// TIA Portal V16 export
// export: Created 2025-08-01T13:38:14.4676832Z, ExportSetting WithDefaults, DisplayName Totally Integrated Automation Portal, DisplayVersion V16, DisplayName TIA Portal Version Control Interface, DisplayVersion V16, DisplayName TIA Portal Openness, DisplayVersion V16, DisplayName STEP 7 Professional, DisplayVersion V16, DisplayName STEP 7 Safety, DisplayVersion V16, DisplayName WinCC Advanced, DisplayVersion V16
VAR_GLOBAL   // PLC tag table "Default tag table"
   "Drive 1 Ready" AT %I0.0 : Bool;   // +MC-21K2:1 - Drive 1 Ready
   "Drive 2 Ready" AT %I0.1 : Bool;   // +MC-21K2:5 - Drive 2 Ready
   "Drive 3 Ready" AT %I0.2 : Bool;   // +MC-21K2:2 - Drive 3 Ready
   "Drive 4 Ready" AT %I0.3 : Bool;   // +MC-21K2:6 - Drive 4 Ready
   "Drive 5 Ready" AT %I0.4 : Bool;   // +MC-21K2:3 - Drive 5 Ready
   "Sensor Trechter" AT %I0.5 : Bool;   // +MC-21K2:7 - Sensor Trechter
   "Sensor Op Band" AT %I0.6 : Bool;   // +MC-21K2:4 Sensor Op Band
   "Sensor Wals (Option)" AT %I0.7 : Bool;   // +MC-21K2:8 - Sensor Wals (Option)
   "ESB Oke" AT %I1.0 : Bool;   // +MC-21K3:1 - ESB Oke
   "ESB Pressend" AT %I1.1 : Bool;   // +MC-21K3:5 - ESB Pressend
   "Reset Active" AT %I1.2 : Bool;   // +MC-21K3:2 - Reset Active
   "Noodsleutel(1)" AT %I1.3 : Bool;   // +MC-21K3:6 - NOODSLEUTEL
   "Alle uitgangen(1)" AT %I1.4 : Bool;   // +MC-21K3:3 - Alle uitgangen
   "Door 1 NC contact" AT %I1.5 : Bool;   // +MC-21K3:7 - Safety Doorswitch 1
   "Door 1 NO contact" AT %I1.6 : Bool;   // +MC-21K3:4 - Safety Doorswitch 1 Normaly open
   "Door 2 NC contact" AT %I1.7 : Bool;   // +MC-21K3:8 - Safety Doorswitch 2
   "Spare(5)" AT %I3.0 : Bool;
   "Spare(6)" AT %I3.1 : Bool;
   "Spare(10)" AT %I180.0 : Bool;   // Spare
   "Spare(11)" AT %I180.1 : Bool;   // Spare
   "Spare(12)" AT %I3.4 : Bool;   // Spare
   "Spare(13)" AT %I3.5 : Bool;   // Spare
   "Spare(14)" AT %I3.6 : Bool;   // Spare
   "Spare(15)" AT %I3.7 : Bool;   // Spare
   "Programma 1" AT %I2.0 : Bool;   // +MC-21K4:1 - Programma 1
   "Programma 2" AT %I2.1 : Bool;   // +MC-21K4:5 - Programma 2 (Option)
   "Programma 3" AT %I2.2 : Bool;   // +MC-21K4:2 - Programma 3
   Cleaning AT %I2.3 : Bool;   // +MC-21K4:6 - Cleaning
   "Start Machine" AT %I2.4 : Bool;   // +MC-21K4:3 - Start Machine
   "Stop Machine" AT %I2.5 : Bool;   // +MC-21K4:7 - Stop Machine
   "Spare(16)" AT %I2.6 : Bool;   // Spare
   Encoder_Z_Puls AT %I2.7 : Bool;   // Spare
   "Safety Relais" AT %Q0.0 : Bool;   // +MC-21K6:1 - Safety Relais
   "Bel Storing" AT %Q0.1 : Bool;   // +MC-21K6:5 - Bel Storing
   Spare AT %Q5.3 : Bool;   // Spare
   "Drive 1 RUN FWD" AT %Q1.0 : Bool;   // +MC-21K8:1 - Drive 1 RUN FWD
   "Drive 1 REV]" AT %Q1.1 : Bool;   // +MC-21K8:5 - Drive 1 REV
   "Drive 1 Speed 1" AT %Q1.2 : Bool;   // +MC-21K8:2 - Drive 1 Speed 1
   "Drive 1 Speed 2" AT %Q1.3 : Bool;   // +MC-21K8:6 - Drive 1 Speed 2
   "Spare(3)" AT %Q1.4 : Bool;   // Spare
   "Drive 2 RUN FWD" AT %Q1.5 : Bool;   // +MC-21K8:7 - Drive 2 RUN FWD
   "Drive 2 REV" AT %Q1.6 : Bool;   // +MC-21K8:4 - Drive 2 REV
   "Drive 2 Speed 1" AT %Q1.7 : Bool;   // +MC-21K8:8 - Drive 2 Speed 1
   "Drive 2 Speed 2" AT %Q2.0 : Bool;   // +MC-21K9:1 - Drive 2 Speed 2
   "Spare(4)" AT %Q2.1 : Bool;   // Spare
   "Drive 3 RUN FWD" AT %Q2.2 : Bool;   // +MC-21K9:2 - Drive 3 RUN FWD
   "Drive 3 REV" AT %Q2.3 : Bool;   // +MC-21K9:6 - Drive 3 REV
   "Drive 3 Speed 1" AT %Q2.4 : Bool;   // +MC-21K9:3 - Drive 3 Speed 1
   "Drive 3 Speed 2" AT %Q2.5 : Bool;   // +MC-21K9:7 - Drive 3 Speed 2
   "Spare(21)" AT %Q2.6 : Bool;   // Spare
   "Drive 4 RUN FWD" AT %Q2.7 : Bool;   // +MC-21K9:8 - Drive 4 RUN FWD
   "Drive 4 REV" AT %Q3.0 : Bool;   // +MC-21K10:1 - Drive 4 REV
   "Drive 4 Speed 1" AT %Q3.1 : Bool;   // +MC-21K10:5 - Drive 4 Speed 1
   "Drive 4 Speed 2" AT %Q3.2 : Bool;   // +MC-21K10:2 - Drive 4 Speed 2
   "Spare(22)" AT %Q3.3 : Bool;   // Spare
   "Drive 5 RUN FWD" AT %Q3.4 : Bool;   // +MC-21K10:3 - Drive 5 RUN FWD
   "Drive 5 REV" AT %Q3.5 : Bool;   // +MC-21K10:7 - Drive 5 REV
   "Drive 5 Speed 1" AT %Q3.6 : Bool;   // +MC-21K10:4 - Drive 5 Speed 1
   "Drive 5 Speed 2" AT %Q3.7 : Bool;   // +MC-21K10:8 - Drive 5 Speed 2
   "Spare(23)" AT %Q4.0 : Bool;   // Spare
   "LED Programma 1" AT %Q4.1 : Bool;   // +MC-21K11:5 - LED Programma 1
   "LED Programma 2" AT %Q4.2 : Bool;   // +MC-21K11:2 - LED Programma 2
   "LED Programma 3" AT %Q4.3 : Bool;   // +MC-21K11:6 - LED Programma 3
   "LED E-STOP" AT %Q0.2 : Bool;   // +MC-21K6:2- LED E-STOP
   "LED RUN" AT %Q4.5 : Bool;   // +MC-21K11:7 - LED RUN
   "Valve 1" AT %Q4.6 : Bool;   // +MC-21K11:4 - Valve 1
   "Valve 2" AT %Q4.7 : Bool;   // +MC-21K11:8 - Valve 2
   "Valve 3" AT %Q5.0 : Bool;   // +MC-21K12:1 - Valve 3
   "Valve 4" AT %Q5.1 : Bool;   // +MC-21K12:5 - Valve 4
   "Valve 5" AT %Q5.2 : Bool;   // +MC-21K12:2 - Valve 5
   "Spare(1)" AT %Q6.0 : Bool;   // Spare
   "Spare(2)" AT %Q6.1 : Bool;   // Spare
   "Spare(18)" AT %Q6.2 : Bool;   // Spare
   "Spare(19)" AT %Q6.3 : Bool;   // Spare
   "Spare(20)" AT %Q4.4 : Bool;   // Spare
   "Drive 1 Rapid Stop" AT %Q0.3 : Bool;   // +MC-21K6:6 - Drive 1 Rapid Stop
   "Drive 2 Rapid Stop" AT %Q0.4 : Bool;   // +MC-21K6:3 - Drive 2 Rapid Stop
   "Drive 3 Rapid Stop" AT %Q0.5 : Bool;   // +MC-21K6:7 - Drive 3 Rapid Stop
   "Drive 4 Rapid Stop" AT %Q0.6 : Bool;   // +MC-21K6:4 - Drive 4 Rapid Stop
   "Drive 5 Rapid Stop" AT %Q0.7 : Bool;   // +MC-21K6:8 - Drive 5 Rapid Stop
   "Systeem RUN" AT %M0.0 : Bool;   // Systeem RUN
   Tag_1 AT %M0.1 : Bool;
   Tag_2 AT %M0.2 : Bool;
   Tag_3 AT %M0.3 : Bool;
   Tag_4 AT %M0.4 : Bool;
   "Safety Feedback" AT %M0.6 : Bool;
   Tag_5 AT %M0.7 : Bool;
   Tag_6 AT %M1.0 : Bool;
   "ONC Drive 1 RUN FWD" AT %M10.0 : Bool;
   "ONC Drive 2 RUN FWD" AT %M10.1 : Bool;
   "ONC Drive 3 RUN FWD" AT %M10.2 : Bool;
   "ONC Drive 4 RUN FWD" AT %M10.3 : Bool;
   "ONC Drive 5 RUN FWD" AT %M10.4 : Bool;
   "ONC Drive 1 RUN FWD and Speed 1" AT %M10.5 : Bool;
   "ONC Drive 2 RUN FWD and Speed 1" AT %M10.6 : Bool;
   "ONC Drive 3 RUN FWD and Speed 1" AT %M10.7 : Bool;
   "ONC Drive 4 RUN FWD and Speed 1" AT %M11.0 : Bool;
   "ONC Drive 5 RUN FWD and Speed 1" AT %M11.1 : Bool;
   "ONC Drive 1 RUN FWD and Speed 2" AT %M11.2 : Bool;
   "ONC Drive 2 RUN FWD and Speed 2" AT %M11.3 : Bool;
   "ONC Drive 3 RUN FWD and Speed 2" AT %M11.4 : Bool;
   "ONC Drive 4 RUN FWD and Speed 2" AT %M11.5 : Bool;
   "ONC Drive 5 RUN FWD and Speed 2" AT %M11.6 : Bool;
   Startknop_Scherm AT %M15.0 : Bool;
   Stopknop_Scherm AT %M15.1 : Bool;
   Tag_7 AT %M110.1 : Bool;
   Reset_scherm AT %M15.2 : Bool;
   Sensor_op_band_memory AT %M15.3 : Bool;
   "System RUN_1" AT %M20.0 : Bool;
   ResetDelay AT %M20.1 : Bool;
   SensorWalsMemory AT %M20.2 : Bool;
   Timer_Memory AT %M20.3 : Bool;
   StopAll AT %M20.4 : Bool;
   Tag_8 AT %M100.3 : Bool;
   Tag_9 AT %M100.4 : Bool;
   Tag_10 AT %M0.5 : Bool;
   Tag_11 AT %M150.0 : Bool;
   Tag_12 AT %M101.1 : Bool;
   Tag_13 AT %T1 : Timer;
   Tag_14 AT %M300.0 : Bool;
   Tag_15 AT %M260.0 : Bool;
   Tag_16 AT %M300.1 : Bool;
   Tag_17 AT %M501.0 : Bool;
   Tag_18 AT %M500.1 : Bool;
   Tag_19 AT %M160.0 : Bool;
   Tag_20 AT %M150.5 : Bool;
   Tag_21 AT %QD256 : DWord;
   Tag_22 AT %QW260 : Word;
   Tag_23 AT %ID256 : DWord;
   Tag_24 AT %ID260 : DWord;
   Tag_25 AT %ID464 : DWord;
   Tag_26 AT %ID471 : DWord;
   Tag_27 AT %QW471 : Word;
   Tag_28 AT %QD464 : DWord;
   Tag_30 AT %IW205 : Int;
   SystemTime AT %MD2 : Time;
   Tag_31 AT %M5.0 : Bool;
   Lamp_Green AT %Q7.0 : Bool;
   Lamp_Blue AT %Q7.1 : Bool;
   Lamp_Yellow AT %Q7.2 : Bool;
   Lamp_Red AT %Q7.3 : Bool;
   Lamp_Buzzer AT %Q7.4 : Bool;
   PulseTimer AT %T0 : Timer;
   Zpuls_Encoder_Band_Set AT %M1.1 : Bool;
   Drive_1_RefRun AT %M1.2 : Bool;
   Tag_32 AT %QD110 : DWord;
   Tag_33 AT %QD111 : DWord;
   Tag_34 AT %QD112 : DWord;
   Tag_35 AT %QD113 : DWord;
   Tag_36 AT %QD114 : DWord;
   Tag_37 AT %QD115 : DWord;
   Tag_38 AT %QD116 : DWord;
   Tag_39 AT %QD117 : DWord;
   Tag_40 AT %QB110 : Byte;
   Tag_41 AT %QB111 : Byte;
   Tag_42 AT %QB112 : Byte;
   Tag_43 AT %QB113 : Byte;
   Tag_44 AT %IB110 : Byte;
   Tag_45 AT %IB111 : Byte;
   Tag_46 AT %IB112 : Byte;
   Tag_47 AT %IB113 : Byte;
   Tag_48 AT %IB114 : Byte;
   Tag_49 AT %IB115 : Byte;
   Tag_50 AT %IB116 : Byte;
   Tag_51 AT %IB117 : Byte;
   Tag_52 AT %QD260 : DWord;
   Tag_53 AT %QB114 : Byte;
   Tag_54 AT %QB115 : Byte;
   Tag_55 AT %QB116 : Byte;
   Tag_56 AT %QB117 : Byte;
   Tag_57 AT %QW256 : Word;
   Tag_58 AT %QW258 : Word;
   Tag_59 AT %IW256 : Word;
   Tag_60 AT %IW258 : Word;
   Tag_61 AT %QW112 : Word;
END_VAR
